FUNCTION_BLOCK FB_INT_UINT (* INT to UINT conversion with limiting *)
  (* Standard: 61499-1-D.1; Classification: Type conversion functions *)
  (* Version 0.0, 2006-06-08, JHC, Holobloc Inc *)
  (* Compiler header: package fb.rt.math; *)
  (* Compiler classdef: class FB_INT_UINT extends FBFunction1 *)
  (* Compiler Java IBM VisualAge 3.0 *)
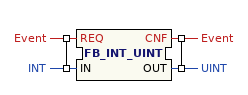
  EVENT_INPUT
    REQ WITH IN;
  END_EVENT
  EVENT_OUTPUT
    CNF WITH OUT;
  END_EVENT
  VAR_INPUT
    IN : INT;
  END_VAR
  VAR_OUTPUT
    OUT : UINT; (* Converted value,-1<OUT<32767 *)
  END_VAR
END_FUNCTION_BLOCK
